ABB RobotStudio station: sesion4_p0.rspag

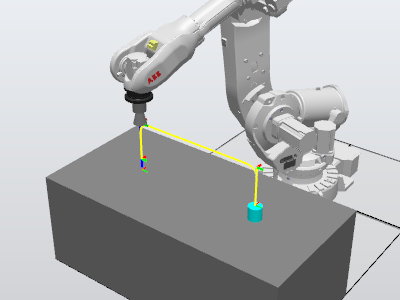
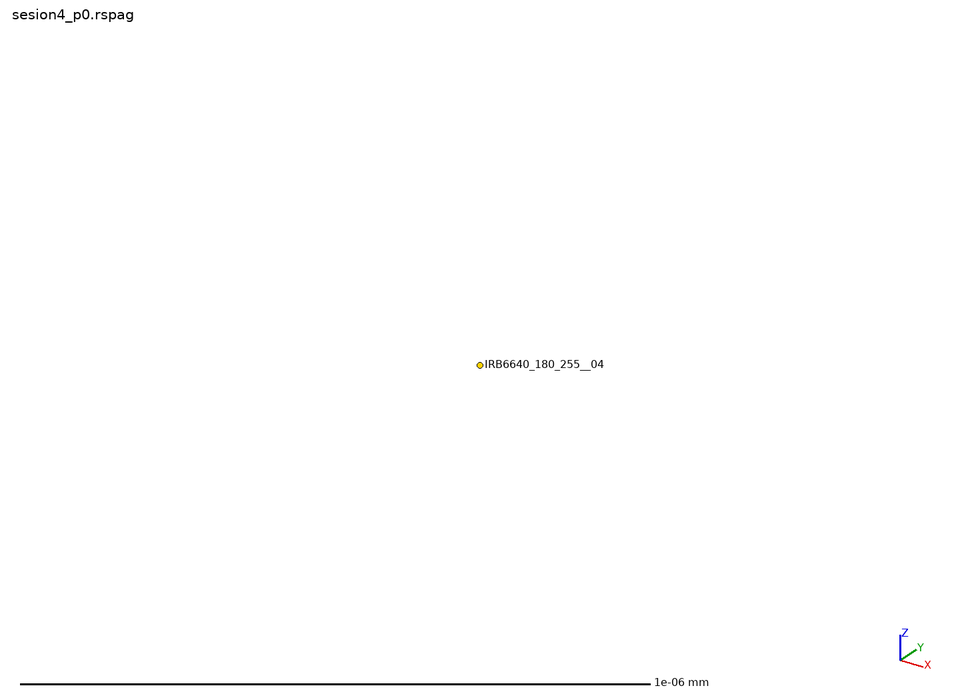
[picture v1: parts stored in the station drawn from their meshes, with robot base, taught points and paths (robot models come from the ABB library and are not in the file)]
--- station ---
Station sesion4 (saved by RobotStudio 24.1.10713.1)
Controller Controlador3
  mechanical unit ROB_1: IRB6640_180_255__04, 6 joints, base frame (0, 0, 0) mm
Layout (positions relative to the parent item):
  - Ventosa [mechanism] at (1500, -500, 1350) mm, rotated rx 180 ry 0 rz 180 deg
      TCP Ventosa at (0, 0, 200) mm
      links: PiezaVentosa
  - IRB6640_180_255__04 [mechanism, from %ABB.RobotStudio.Models.IRB6640%\IRB6640_180_255_G_04.rslib] at (0, 0, 0) mm; joint values [-0.3218, 0.1303, 0.301, 0, 1.1395, -0.3218] (rad or m)
  - Pieza_4 [part], size 1000 x 1000 x 750 mm
  - Pieza_5 [part], size 1000 x 1000 x 750 mm
  - Pieza_6 [part], size 100 x 99.8 x 100 mm
Attachment: Ventosa is attached to IRB6640_180_255__04 / Link6
Targets, tools, work objects and paths stored in the station and not in the controller backup, written as RAPID:
! task T_ROB1
MODULE CalibData
  PERS tooldata Ventosa:=[TRUE,[[0,0,200],[1,0,0,0]],[1,[0,0,125],[1,0,0,0],0.002,0.002,0.0013]];
ENDMODULE

! task T_ROB1
MODULE Module1
  CONST robtarget pBaseOrigen:=[[1500,500,750],[0,0,1,0],[0,0,0,0],[9E+09,9E+09,9E+09,9E+09,9E+09,9E+09]];
  CONST robtarget pBaseDestino:=[[1500,-500,750],[0,0,1,0],[0,0,0,0],[9E+09,9E+09,9E+09,9E+09,9E+09,9E+09]];
  CONST robtarget pOrigen:=[[1500,500,850],[0,0,1,0],[0,0,0,0],[9E+09,9E+09,9E+09,9E+09,9E+09,9E+09]];
  CONST robtarget pDestino:=[[1500,-500,850],[0,0,1,0],[-1,0,-1,0],[9E+09,9E+09,9E+09,9E+09,9E+09,9E+09]];
  CONST robtarget pOrigenAprox:=[[1500,500,1150],[0,0,1,0],[0,0,0,0],[9E+09,9E+09,9E+09,9E+09,9E+09,9E+09]];
  CONST robtarget pDestinoAprox:=[[1500.000049807,-500.000011712,1150.000037959],[-0.000000035,0.000000015,1,0.000000012],[-1,-1,-1,0],[9E+09,9E+09,9E+09,9E+09,9E+09,9E+09]];
  PROC Path_10()
    MoveJ pOrigenAprox,v1000,z100,Ventosa\WObj:=wobj0;
    MoveL pOrigen,v400,fine,Ventosa\WObj:=wobj0;
    MoveL pOrigenAprox,v400,z100,Ventosa\WObj:=wobj0;
    MoveL pDestinoAprox,v2000,z100,Ventosa\WObj:=wobj0;
    MoveL pDestino,v400,fine,Ventosa\WObj:=wobj0;
    MoveL pDestinoAprox,v400,fine,Ventosa\WObj:=wobj0;
  ENDPROC
ENDMODULE


--- Backups/Controlador3/RAPID/TASK1/PROGMOD/Module1.mod ---
MODULE Module1
    !***********************************************************
    !
    ! M?dulo:  Module1
    !
    ! Descripción:
    !   <Introduzca la descripción aquí>
    !
    ! Autor: yisus
    !
    ! Versión: 1.0
    !
    !***********************************************************


    !***********************************************************
    !
    ! Procedimiento Main
    !
    !   Este es el punto de entrada de su programa
    !
    !***********************************************************
    PROC main()
        !Add your code here
    ENDPROC
ENDMODULE

--- Backups/Controlador3/SYSPAR/EIO.cfg ---
EIO:CFG_1.0:6:1::
#
INDUSTRIAL_NETWORK:

      -Name "DeviceNet" -Label "DeviceNet Master/Slave Network" -Address "2"
#
DEVICENET_INTERNAL_DEVICE:

      -Name "DN_Internal_Device" -VendorName "ABB Robotics"\
      -ProductName "DeviceNet Internal Slave Device"
